{attribute 'no_explicit_call' := 'Do not call this function block directly. Please use the provided methods.'} 
FUNCTION_BLOCK FINAL TcoArguments IMPLEMENTS ITcoArguments
VAR
	_data			: ARRAY[0.. (MAX_ARGUMENTS - 1)] OF T_Arg;
	_count			: UINT;
	_ipLogger		: ITcoLogger;
END_VAR


VAR CONSTANT
	MAX_ARGUMENTS	: USINT := 10;
END_VAR

METHOD AddBool : ITcoArguments
VAR_INPUT
	Value		: BOOL;
END_VAR
IF _count < MAX_ARGUMENTS THEN
	_data[_count] := F_BOOL(Value);
	_count := _count + 1;
END_IF

AddBool := THIS^;
END_METHOD

METHOD AddDecimal : ITcoArguments
VAR_INPUT
	Value	: DINT;
END_VAR
IF _count < MAX_ARGUMENTS THEN
	_data[_count] := F_DINT(Value);
	_count := _count + 1;
END_IF

AddDecimal := THIS^;
END_METHOD

METHOD AddFloat : ITcoArguments
VAR_INPUT
	Value	: LREAL;
END_VAR
IF _count < MAX_ARGUMENTS THEN
	_data[_count] := F_LREAL(Value);
	_count := _count + 1;
END_IF

AddFloat := THIS^;
END_METHOD

METHOD AddString : ITcoArguments
VAR_INPUT
	Value	: STRING;
END_VAR
IF _count < MAX_ARGUMENTS THEN
	_data[_count] := F_STRING(Value);
	_count := _count + 1;
END_IF

AddString := THIS^;
END_METHOD

METHOD AddStruct : ITcoArguments
VAR_INPUT
	(*~
	<docu>
		<summary>
			Size of the variable. Is typicaly determined by `SIZEOF` opreator: SIZEOF(Variable)
		</summary>				
	</docu>	
	~*)
	ioSIZE : UDINT;
	(*~
	<docu>
		<summary>
			Pointer to the variable is typically determined by `ADR` operator ADR(Variable)
		</summary>				
	</docu>	
	~*)
	pVARIABLE : POINTER TO ULINT;
END_VAR


VAR
	jsonConverter 	: Tc3_JsonXml.FB_JsonReadWriteDatatype;	
	jsonDoc			: STRING(255);
	jsonDocSize		: UDINT := SIZEOF(jsonDoc);
	symbolName		: STRING(255);
	arg				: T_Arg;
END_VAR
IF pVARIABLE <> 0 AND ioSIZE > 0 AND _count < MAX_ARGUMENTS THEN
	symbolName := jsonConverter.GetSymbolNameByAddress(nData := ioSIZE, pData := pVARIABLE);
	
	IF jsonConverter.GetJsonFromSymbol(symbolName, ioSIZE, pVARIABLE, jsonDocSize, jsonDoc) THEN
		
		arg.eType := ARGTYPE_STRING;
		arg.cbLen := INT_TO_UDINT( LEN2( ADR(jsonDoc) ) + 1 );
		arg.pData := pVARIABLE;
	
		_data[_count] := arg;
		_count := _count + 1;
	
	END_IF
END_IF

AddStruct := THIS^;
END_METHOD

METHOD Append : ITcoLogger
Append := _ipLogger;
END_METHOD

METHOD Clear : ITcoArguments
MEMSET(ADR(_data), 0, SIZEOF(_data));
Clear := THIS^;
END_METHOD

METHOD PUBLIC Compose : BOOL
VAR_INPUT
	Message		: POINTER TO STRING(255);
END_VAR


VAR
	messageFormatter		: Tc2_Utilities.FB_FormatString2;
END_VAR
// format specification
// https://infosys.beckhoff.com/english.php?content=../content/1033/tcplclib_tc2_utilities/35403019.html&id=5274291506655699832

messageFormatter(
	pFormatString	:= Message, 
	arg1			:= _data[0], 
	arg2			:= _data[1], 
	arg3			:= _data[2], 
	arg4			:= _data[3], 
	arg5			:= _data[4], 
	arg6			:= _data[5], 
	arg7			:= _data[6], 
	arg8			:= _data[7], 
	arg9			:= _data[8], 
	arg10			:= _data[9],
	pDstString		:= Message, 
	nDstSize		:= SIZEOF(Message));
	
Compose := NOT messageFormatter.bError;
END_METHOD

METHOD FB_init : BOOL
VAR_INPUT
	bInitRetains : BOOL; // if TRUE, the retain variables are initialized (warm start / cold start)
	bInCopyCode : BOOL;  // if TRUE, the instance afterwards gets moved into the copy code (online change)
	
	Logger		: ITcoLogger;
END_VAR
_ipLogger := Logger;
END_METHOD

PROPERTY PUBLIC IsEmpty : BOOL
GET
IsEmpty := _count = 0;
END_GET
END_PROPERTY

END_FUNCTION_BLOCK

(* stored: Version 1.1.0.1, ProductVersion 3.1.4024.9
   POU TcoArguments: Id {1e14562d-c399-070d-1868-6b15d94c6a55}, SpecialFunc None
   Method AddBool: Id {cb64d28d-ed40-0f31-241d-5d73544c21ed}
   Method AddDecimal: Id {50aa3f44-94cd-0023-344f-6679e7c2164f}
   Method AddFloat: Id {0d76284b-3238-0556-091b-f4b9e1cdea7e}
   Method AddString: Id {2474d8f9-ade5-0a8d-2f75-95232d506eb4}
   Method AddStruct: Id {ba40cb5d-f986-0d3b-0d1d-d5d746da8b89}
   Method Append: Id {30f30573-bcb2-0fb3-3b74-7e220ac0b12f}
   Method Clear: Id {9d22b885-9d89-08cb-06fc-dd69d845abfc}
   Method Compose: Id {9f09b9de-8020-0eb7-2099-0f2b40d01b4b}
   Method FB_init: Id {1f656fc0-0ad8-0b1c-00b4-36109accc461}
   Property IsEmpty: Id {2efba640-4f4d-05de-2f84-69bf90243d91}
   Get Get: Id {598f0cfb-bb4d-0e68-1a16-b2f834a2db2e} *)
